FUNCTION_BLOCK MOVING_AVERAGE_V2
  {SET_ATTRIBUTE(OpcUa, SERVICE)}
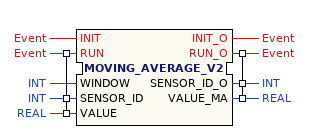
  EVENT_INPUT
    INIT;
    RUN WITH VALUE, SENSOR_ID; {SET_ATTRIBUTE(OpcUa, Method)}
  END_EVENT
  EVENT_OUTPUT
    INIT_O;
    RUN_O WITH VALUE_MA, SENSOR_ID_O;
  END_EVENT
  VAR_INPUT
    WINDOW : INT; {SET_ATTRIBUTE(OpcUa, Constant.RUN)}
    SENSOR_ID : INT; {SET_ATTRIBUTE(OpcUa, Variable.RUN)}
    VALUE : REAL; {SET_ATTRIBUTE(OpcUa, Variable.RUN)}
  END_VAR
  VAR_OUTPUT
    SENSOR_ID_O : INT; {SET_ATTRIBUTE(OpcUa, Variable.RUN)}
    VALUE_MA : REAL; {SET_ATTRIBUTE(OpcUa, Variable.RUN)}
  END_VAR
END_FUNCTION_BLOCK
